DATA_BLOCK "output"
{ S7_Optimized_Access := 'FALSE' }
VERSION : 0.1
NON_RETAIN
   STRUCT
      "1层上行呼梯按钮指示灯" : Bool;
      "2层上行呼梯按钮指示灯" : Bool;
      "3层上行呼梯按钮指示灯" : Bool;
      "4层上行呼梯按钮指示灯" : Bool;
      "5层上行呼梯按钮指示灯" : Bool;
      "2层下行呼梯按钮指示灯" : Bool;
      "3层下行呼梯按钮指示灯" : Bool;
      "4层下行呼梯按钮指示灯" : Bool;
      "5层下行呼梯按钮指示灯" : Bool;
      "6层下行呼梯按钮指示灯" : Bool;
      "1号梯1层按钮指示灯" : Bool;
      "1号梯2层按钮指示灯" : Bool;
      "1号梯3层按钮指示灯" : Bool;
      "1号梯4层按钮指示灯" : Bool;
      "1号梯5层按钮指示灯" : Bool;
      "1号梯6层按钮指示灯" : Bool;
      "1号梯LEDa" : Bool;
      "1号梯LEDb" : Bool;
      "1号梯LEDc" : Bool;
      "1号梯LEDd" : Bool;
      "1号梯LEDe" : Bool;
      "1号梯LEDf" : Bool;
      "1号梯LEDg" : Bool;
      "1号梯上行指示" : Bool;
      "1号梯下行指示" : Bool;
      "1号梯故障指示" : Bool;
      "1号梯照明指示" : Bool;
      "1号梯风扇指示" : Bool;
      "1号梯满载指示" : Bool;
      "1号梯电机启动信号" : Bool;
      "1号梯上行接触器" : Bool;
      "1号梯下行接触器" : Bool;
      "1号梯高速接触器" : Bool;
      "1号梯低速接触器" : Bool;
      "1号梯开门继电器" : Bool;
      "1号梯关门继电器" : Bool;
      "1号梯1级减速制动" : Bool;
      "1号梯2级减速制动" : Bool;
      "1号梯3级减速制动" : Bool;
      准备就绪信号 : Bool;
   END_STRUCT;


BEGIN

END_DATA_BLOCK

